{attribute 'qualified_only'}
{attribute 'strict'}
{attribute 'to_string'}
TYPE E_DS402MotionState :
(
    PREPARE_MOTION_PARAMS:=0,
    INITIATE_MOTION:=10,
    DRIVE_IN_MOTION :=20,
    TARGET_REACHED:=30,
	INTERRUPTED:=40,
	ABORTED:=50,
    DONE:=60,
    ERROR:=99
);
END_TYPE

(* stored: Version 1.1.0.1
   DUT E_DS402MotionState: Id {c62d474f-9328-4cf8-a11d-ca4c197acefc} *)
